{attribute addProperty BoxType "EL3773-0000-0018"}
{attribute addProperty Id "U1_StatusAT %I*U1_Status_E2EFACF1162"}
{attribute addProperty CRC "3280589885"}
{attribute addProperty SizeInBites "16"}
{attribute addProperty SizeInBytes "2"}
TYPE L1_Voltage_Status_C389D43D :
STRUCT
	{attribute addProperty Name "U1_Status"}
	U1_Status AT %I* : U1_Status_E2EFACF1;
END_STRUCT
END_TYPE

(* stored: Version 1.2.0.0, ProductVersion 3.1.4024.9
   DUT L1_Voltage_Status_C389D43D: Id {faaeb5f2-0618-423f-9455-71b007ed4825} *)
